// TwinCAT 3 PLC project IntegrationProjects
// Title: IntegrationProjects
// Company: Vortex.Library
// ProjectVersion: 0.6.0.913
// ProgramVersion: 3.1.4023.0
// libraries:
//   Tc2_Standard, * (Beckhoff Automation GmbH)
//   Tc2_System, * (Beckhoff Automation GmbH)
//   Tc3_Module, * (Beckhoff Automation GmbH)
//   TcoCore, 0.6.0.913 (Vortex.Library)
//   TcoData, 0.6.0.913 (Vortex.Library)
//   TcoDrivesBeckhoff, 0.6.0.913 (Vortex.Library)
//   TcoElements, 0.6.0.913 (Vortex.Library)
//   TcoIo, 0.6.0.913 (Vortex.Library)
//   TcoPneumatics, 0.6.0.913 (Vortex.Library)
//   TcoUtilities, 0.6.0.913 (Vortex.Library)
// project tree:
//   / PlcTask.TcTTO
//   POUs/ MAIN.TcPOU, SampleContext.TcPOU
//   POUs/SampleComponent/ SampleComponent.TcPOU, SampleTaskFunctionBuffer.TcDUT, SampleTaskIteration.TcPOU
//   Technology/IO/ EC001.TcDUT, IO.TcGVL
//   Technology/ MAIN_TECHNOLOGY.TcPOU, Technology.TcPOU
//   Technology/ST001/Data/ ST001_ProcessData.TcDUT, ST001_ProcessDataManager.TcPOU
//   Technology/ST001/ ST001.TcPOU, ST001_Components.TcDUT, ST001_ComponentsHandler.TcPOU, ST001_GroundSequence.TcPOU, ST001_AutomatSequence.TcPOU
//   ToLibs/BeckhoffIo/EL1008/ EL1008.TcPOU, EL1008_Data.TcDUT
//   ToLibs/BeckhoffIo/EL2008/ EL2008.TcPOU, EL2008_Data.TcDUT
//   ToLibs/BeckhoffIo/ WcState.TcDUT, InfoData.TcDUT
// real-time tasks:
//   TASK PlcTask: cycle T#10ms, priority 20, ADS port 350
//   TASK PlcTask1: cycle T#10ms, priority 21, ADS port 351
// I/O:
//   DEVICE Device 1 (EtherCAT) (disabled), AmsNetId 172.20.10.104.2.1
//     EC001 (EK1100) [EK1100 EtherCAT Coupler (2A E-Bus)]
//       A1 (EL1008) [EL1008 8Ch. Dig. Input 24V, 3ms]
//       A10 (EL2008) [EL2008 8Ch. Dig. Output 24V, 0.5A]

CONFIGURATION IntegrationProjects
    RESOURCE PLC ON TwinCAT3
        TASK PlcTask(INTERVAL := T#10ms, PRIORITY := 20);
        PROGRAM MAIN WITH PlcTask : MAIN;
        PROGRAM MAIN_TECHNOLOGY WITH PlcTask : MAIN_TECHNOLOGY;
    END_RESOURCE
END_CONFIGURATION

// ---- POUs/SampleComponent/SampleTaskFunctionBuffer.TcDUT
TYPE SampleTaskFunctionBuffer :
    STRUCT
    x : LREAL;
    y : LREAL;
END_STRUCT
END_TYPE

// ---- Technology/IO/EC001.TcDUT
TYPE EC001 :
    STRUCT
    {attribute addProperty Name "A1"}
    A1 : EL1008;
    {attribute addProperty Name "A10"}
    A10 : EL2008;
END_STRUCT
END_TYPE

// ---- Technology/ST001/Data/ST001_ProcessData.TcDUT
TYPE ST001_ProcessData EXTENDS TcoData.TcoEntity :
STRUCT
    PressingTime : TIME;
END_STRUCT
END_TYPE

// ---- Technology/ST001/ST001_Components.TcDUT
TYPE ST001_Components :
    STRUCT
    PartPresent : TcoElements.TcoDi(MAIN_TECHNOLOGY._technology._ST001);
    StartButton : TcoElements.TcoDi(MAIN_TECHNOLOGY._technology._ST001);
    Press : TcoPneumatics.TcoCylinder(MAIN_TECHNOLOGY._technology._ST001);
    Drive : TcoDriveSimple(MAIN_TECHNOLOGY._technology._ST001);
END_STRUCT
END_TYPE

// ---- ToLibs/BeckhoffIo/EL1008/EL1008_Data.TcDUT
TYPE EL1008_Data :
STRUCT
    {attribute addProperty Name "1"}
    _1 AT %I* : BOOL;
    {attribute addProperty Name "2"}
    _2 AT %I* : BOOL;
    {attribute addProperty Name "3"}
    _3 AT %I* : BOOL;
    {attribute addProperty Name "4"}
    _4 AT %I* : BOOL;
    {attribute addProperty Name "5"}
    _5 AT %I* : BOOL;
    {attribute addProperty Name "6"}
    _6 AT %I* : BOOL;
    {attribute addProperty Name "7"}
    _7 AT %I* : BOOL;
    {attribute addProperty Name "7"}
    _8 AT %I* : BOOL;
    WcState : WcState;
    InfoData : InfoData;
END_STRUCT
END_TYPE

// ---- ToLibs/BeckhoffIo/EL2008/EL2008_Data.TcDUT
TYPE EL2008_Data :
STRUCT
    {attribute addProperty Name "1"}
    _1 AT %Q* : BOOL;
    {attribute addProperty Name "2"}
    _2 AT %Q* : BOOL;
    {attribute addProperty Name "3"}
    _3 AT %Q* : BOOL;
    {attribute addProperty Name "4"}
    _4 AT %Q* : BOOL;
    {attribute addProperty Name "5"}
    _5 AT %Q* : BOOL;
    {attribute addProperty Name "6"}
    _6 AT %Q* : BOOL;
    {attribute addProperty Name "7"}
    _7 AT %Q* : BOOL;
    {attribute addProperty Name "8"}
    _8 AT %Q* : BOOL;
    WcState : WcState;
    InfoData : InfoData;
END_STRUCT
END_TYPE

// ---- ToLibs/BeckhoffIo/WcState.TcDUT
TYPE WcState :
STRUCT
    State AT %I* : BOOL;
    InputToggle AT %I* : BOOL;
END_STRUCT
END_TYPE

// ---- ToLibs/BeckhoffIo/InfoData.TcDUT
TYPE InfoData :
STRUCT
    State AT %I* : UINT;
END_STRUCT
END_TYPE

// ---- Technology/IO/IO.TcGVL
{attribute 'qualified_only'}
VAR_GLOBAL
    {attribute addProperty Name "EC001"}
    EC001 : EC001;
END_VAR

// ---- POUs/MAIN.TcPOU
PROGRAM MAIN
VAR
    _sampleContext : SampleContext;
END_VAR

_sampleContext.Run();

END_PROGRAM

// ---- POUs/SampleContext.TcPOU
FUNCTION_BLOCK SampleContext EXTENDS TcoCore.TcoContext
VAR
    _sampleComponent : SampleComponent(THIS^);
END_VAR

(*~
    <docu>
        <summary>
            Main method of the TcoContext. This is the entry point of any control logic that belongs to this context.
            The call of this method is ensured by calling the <c>InstanceName.Run()</c> method, and it must not be called explicitly.
            This method is abstract, and it must be overridden in derived block.
        </summary>
    </docu>
~*)
METHOD PROTECTED Main
_sampleComponent.Service();
_sampleComponent();
END_METHOD

END_FUNCTION_BLOCK

// ---- POUs/SampleComponent/SampleComponent.TcPOU
(*~
    <docu>
        <summary>Sample component for inspiration</summary>
    </docu>
~*)
FUNCTION_BLOCK SampleComponent EXTENDS TcoCore.TcoComponent
VAR
    (*~
        <docu>
            <summary>Counter</summary>
            <remarks>
                > [!IMPORTANT]
                > This member is ignored when rendering.
            </remarks>
        </docu>
    ~*)
    {attribute clr [RenderIgnore()]}
    _counter : INT;
END_VAR
VAR
    (*~
        <docu>
            <summary>Counter</summary>
            <remarks>
                > [!IMPORTANT]
                > This member is readonly.
            </remarks>
        </docu>
    ~*)
    {attribute addProperty Name "Add Result"}
    {attribute clr [ReadOnly()]}
    _addResult : INT;
    {attribute addProperty Name "A"}
    _addNumberOne : INT;
    {attribute addProperty Name "B"}
    _addNumberTwo : INT;
END_VAR
VAR
    _sampleTask : SampleTaskIteration(THIS^);
END_VAR

_addResult := THIS^.AddTwoNumbers(_addNumberOne, _addNumberTwo);
_sampleTask();

(*~
    <docu>
        <summary>Adds two numbers</summary>
        <returns>Sum of two numbers</returns>
    </docu>
~*)
METHOD AddTwoNumbers : INT
VAR_INPUT
    NumberOne : INT;
    NumberTwo : INT;
END_VAR
AddTwoNumbers := NumberOne + NumberTwo;
END_METHOD

{attribute 'TcRpcEnable'}
METHOD INTERNAL AddTwoNumbersTest : INT
VAR_INPUT
    NumberOne : INT;
    NumberTwo : INT;
END_VAR
AddTwoNumbersTest := THIS^.AddTwoNumbers(NumberOne, NumberTwo);
END_METHOD

METHOD FB_init : BOOL
VAR_INPUT
    bInitRetains : BOOL; // if TRUE, the retain variables are initialized (warm start / cold start)
    bInCopyCode : BOOL; // if TRUE, the instance afterwards gets moved into the copy code (online change)
    ParentObject : ITcoObject;
END_VAR
END_METHOD

(*~
    <docu>
        <summary>
            Restores this instance to the Ready state. Can be called explicitly or from within one of the restore mechanisms.
        </summary>
    </docu>
~*)
METHOD Restore : ITcoRestorable
END_METHOD

(*~
    <docu>
        <summary>
            Custom service (manual, maintenance) logic.
            This method must be implemented in derived class.
        </summary>
    </docu>
~*)
METHOD PROTECTED ServiceMode
END_METHOD

METHOD WaitForModulo : BOOL
VAR_INPUT
    Modulo : INT;
END_VAR
_counter := _counter + 1;
WaitForModulo := _counter MOD Modulo = 0;
END_METHOD

{attribute 'TcRpcEnable'}
METHOD INTERNAL WaitForModuloTest : BOOL
VAR_INPUT
    Modulo : INT;
END_VAR
WaitForModuloTest := THIS^.WaitForModulo(Modulo);
END_METHOD

END_FUNCTION_BLOCK

// ---- POUs/SampleComponent/SampleTaskIteration.TcPOU
FUNCTION_BLOCK SampleTaskIteration EXTENDS TcoCore.TcoTask
VAR
    _x : LREAL;
    _y : LREAL;
    _d : LREAL;
    {attribute addProperty Minimum 100}
    {attribute addProperty Maximum 1000}
    _iterations : INT;
    _currentIteration : INT;
END_VAR

IF (Execute()) THEN
    _y := SIN(_x);
    _x := _x + _d;
    _currentIteration := _currentIteration + 1;
    DoneWhen(_currentIteration >= _iterations);
END_IF

METHOD FB_init : BOOL
VAR_INPUT
    bInitRetains : BOOL; // if TRUE, the retain variables are initialized (warm start / cold start)
    bInCopyCode : BOOL; // if TRUE, the instance afterwards gets moved into the copy code (online change)
    ParentObject : ITcoObject;
END_VAR
END_METHOD

(*~
    <docu>
        <summary>
            Restores this instance to the Ready state. Can be called explicitly or from within one of the restore mechanisms.
            <para>
                See also <see cref="PlcDocu.TcoCore.TcoTask.AutoRestorable()"/>
            </para>
        </summary>
    </docu>
~*)
METHOD Restore : ITcoRestorable
SUPER^.Restore();
_x := 0.0;
_y := 0.0;
_currentIteration := 0;
END_METHOD

END_FUNCTION_BLOCK

// ---- Technology/MAIN_TECHNOLOGY.TcPOU
PROGRAM MAIN_TECHNOLOGY
VAR
    _technology : Technology;
END_VAR

_technology.Run();

END_PROGRAM

// ---- Technology/Technology.TcPOU
FUNCTION_BLOCK Technology EXTENDS TcoCore.TcoContext
VAR
    _ST001 : ST001(THIS^);
    _mirrorStartCycle : ULINT;
END_VAR

(*~
    <docu>
        <summary>
            Main method of the TcoContext. This is the entry point of any control logic that belongs to this context.
            The call of this method is ensured by calling the <c>InstanceName.Run()</c> method, and it must not be called explicitly.
            This method is abstract, and it must be overridden in derived block.
        </summary>
    </docu>
~*)
METHOD PROTECTED Main
_ST001();
END_METHOD

END_FUNCTION_BLOCK

// ---- Technology/ST001/ST001.TcPOU
FUNCTION_BLOCK ST001 EXTENDS TcoCore.TcoObject
VAR
    {attribute addProperty Name "<#MANUAL#>"}
    _serviceModeTask : TcoCore.TcoTask(THIS^);
    {attribute addProperty Name "<#GROUND#>"}
    _groundSequenceTask : TcoCore.TcoTask(THIS^);
    {attribute addProperty Name "<#AUTOMAT#>"}
    _automatSequenceTask : TcoCore.TcoTask(THIS^);
    {attribute clr [Container(Layout.Stack)]}
    _components : ST001_ComponentsHandler(THIS^);
    {attribute clr [RenderIgnore()]}
    _mqttMirrorComponents : ST001_ComponentsHandler(THIS^);
    {attribute clr [Container(Layout.Stack)]}
    _groundPositionSequence : ST001_GroundSequence(THIS^, eRestoreMode.None);
    _automatPositionSequence : ST001_AutomatSequence(THIS^, eRestoreMode.None);
    _settings : ST001_ProcessDataManager(THIS^);
    _repository : ST001_ProcessDataManager(THIS^);
END_VAR

_components();
_settings();
_repository();
_groundPositionSequence(inoComponents := _components);
_automatPositionSequence(inoComponents := _components);

IF (_groundSequenceTask.Execute()) THEN
    _serviceModeTask.Abort();
    _groundPositionSequence.Run();
    _groundSequenceTask.DoneWhen(_groundPositionSequence.CurrentStep.ID = _groundPositionSequence.MaxStepID - 1);
END_IF

_automatSequenceTask.Enabled := _groundSequenceTask.Done;

IF (_automatSequenceTask.Execute()) THEN
    _automatPositionSequence.Run();
END_IF

IF (_serviceModeTask.Execute()) THEN
    _automatSequenceTask.Restore();
    _groundSequenceTask.Restore();
    _groundPositionSequence.Restore();
    _components.Service();
END_IF

PROPERTY Repository : REFERENCE TO ST001_ProcessDataManager
GET
Repository REF= _repository;
END_GET
END_PROPERTY

PROPERTY Settings : REFERENCE TO ST001_ProcessDataManager
GET
Settings REF= _settings;
END_GET
END_PROPERTY

END_FUNCTION_BLOCK

// ---- Technology/ST001/ST001_ComponentsHandler.TcPOU
FUNCTION_BLOCK ST001_ComponentsHandler EXTENDS TcoCore.TcoObject
VAR
    ToMirror : STRING;
    {attribute addProperty Name "<#PART PRESENCE SENSOR#>"}
    _partPresent : TcoElements.TcoDi(THIS^);
    {attribute addProperty Name "<#START BUTTON#>"}
    _startButton : TcoElements.TcoDi(THIS^);
    {attribute addProperty Name "<#PRESS PISTON#>"}
    _press : TcoPneumatics.TcoCylinder(THIS^);
    {attribute addProperty Name "<#ALARM OUTPUT#>"}
    _alarmOutput : TcoElements.TcoDo(THIS^);
    {attribute addProperty Name "<#DRIVE#>"}
    _drive : TcoDrivesBeckhoff.TcoDriveSimple(THIS^);
END_VAR

_partPresent(inoSignal := IO.EC001.A1.IO._1);
_startButton(inoSignal := IO.EC001.A1.IO._2);

_press(inoAtHomePos := IO.EC001.A1.IO._3,
    inoAtWorkPos := IO.EC001.A1.IO._4,
    inoToHomePos := IO.EC001.A10.IO._1,
    inoToWorkPos := IO.EC001.A10.IO._2);

PROPERTY PartPresent : REFERENCE TO TcoElements.TcoDi
GET
PartPresent REF= _partPresent;
END_GET
END_PROPERTY

PROPERTY Press : REFERENCE TO TcoPneumatics.TcoCylinder
GET
Press REF= _press;
END_GET
END_PROPERTY

METHOD Service
THIS^._partPresent.Service();
THIS^._startButton.Service();
THIS^._press.Service();
THIS^._alarmOutput.Service();
END_METHOD

END_FUNCTION_BLOCK

// ---- Technology/ST001/ST001_GroundSequence.TcPOU
FUNCTION_BLOCK ST001_GroundSequence EXTENDS TcoCore.TcoSequencer
VAR_IN_OUT
    inoComponents : ST001_ComponentsHandler;
END_VAR

(*~
    <docu>
        <summary>
            Main method of the sequener. Custom code needs to be placed here. The sequencer is executed by call of InstanceName.Run() method.
            This method is abstract, and it must be overridden in derived block.
        </summary>
    </docu>
~*)
METHOD PROTECTED Main : BOOL
IF (NOT __ISVALIDREF(inoComponents)) THEN
    Messenger.Programming('Invalid reference to inoComponents');
    RETURN;
END_IF

IF (Step(inStepID := 100, inEnabled := TRUE, inStepDescription := '<#PRESS IN BASE POSITION#>')) THEN
    //---------------------------------------
    IF (inoComponents.Press.MoveToHome().Done) THEN
        THIS^.CompleteStep();
    END_IF;
    //---------------------------------------
END_IF;

IF (Step(inStepID := 200, inEnabled := TRUE, inStepDescription := '<#CHECK PART REMOVAL FROM THE FIXTURE#>')) THEN
    //---------------------------------------
    IF (inoComponents.PartPresent.IsFalse) THEN
        THIS^.CompleteStep();
    ELSE
        Messenger.Notify('<#Remove part from the fixture please#>');
    END_IF;
    //---------------------------------------
END_IF;

IF (Step(inStepID := MaxStepID - 1, inEnabled := TRUE, inStepDescription := '<#GROUND POSITION COMPLETED#>')) THEN
    //---------------------------------------
    Messenger.Notify('<#Ground position completed; you can start automat sequence.#>');
    //---------------------------------------
END_IF;
END_METHOD

METHOD PROTECTED OnStateChange
VAR_INPUT
    PreviousState : INT;
    NewState : INT;
END_VAR
IF (NOT __ISVALIDREF(inoComponents)) THEN
    RETURN;
END_IF

inoComponents.Press.Restore();
END_METHOD

END_FUNCTION_BLOCK

// ---- Technology/ST001/ST001_AutomatSequence.TcPOU
FUNCTION_BLOCK ST001_AutomatSequence EXTENDS TcoCore.TcoSequencer
VAR_IN_OUT
    inoComponents : ST001_ComponentsHandler;
END_VAR
VAR
    _gTimer_1 : Tc2_Standard.TON;
END_VAR

(*~
    <docu>
        <summary>
            Main method of the sequener. Custom code needs to be placed here. The sequencer is executed by call of InstanceName.Run() method.
            This method is abstract, and it must be overridden in derived block.
        </summary>
    </docu>
~*)
METHOD PROTECTED Main : BOOL
IF (NOT __ISVALIDREF(inoComponents)) THEN
    Messenger.Programming('Invalid reference to inoComponents');
    RETURN;
END_IF

IF (Step(inStepID := 100, inEnabled := TRUE, inStepDescription := '<#LOAD PART INTO FIXTURE#>')) THEN
    //---------------------------------------
    IF (inoComponents.PartPresent.IsTrue) THEN
        THIS^.CompleteStep();
    END_IF;
    //---------------------------------------
END_IF;

IF (Step(inStepID := 200, inEnabled := TRUE, inStepDescription := '<#PRESS START BUTTON TO START OPERATIONS#>')) THEN
    //---------------------------------------
    IF (inoComponents._startButton.IsTrue) THEN
        THIS^.CompleteStep();
    END_IF;
    //---------------------------------------
END_IF;

IF (Step(inStepID := 300, inEnabled := TRUE, inStepDescription := '<#PRESSING#>')) THEN
    //---------------------------------------
    _gTimer_1(IN := inoComponents.Press.MoveToWork().Done, PT := T#500MS);

    IF (_gTimer_1.Q) THEN
        THIS^.CompleteStep();
    END_IF;
    //---------------------------------------
END_IF;

IF (Step(inStepID := 400, inEnabled := TRUE, inStepDescription := '<#MOVING PRESS TO HOME POSITION#>')) THEN
    //---------------------------------------
    IF (inoComponents.Press.MoveToHome().Done) THEN
        THIS^.CompleteStep();
    END_IF;
    //---------------------------------------
END_IF;

IF (Step(inStepID := 500, inEnabled := TRUE, inStepDescription := '<#REMOVE PART FROM THE FIXTURE#>')) THEN
    //---------------------------------------
    IF (inoComponents.PartPresent.IsFalse) THEN
        THIS^.CompleteStep();
    END_IF;
    //---------------------------------------
END_IF;

IF (Step(inStepID := 600, inEnabled := TRUE, inStepDescription := '<#SAVE DATA#>')) THEN
    //---------------------------------------
    IF (THIS^.Station^.Settings.Create(ULINT_TO_STRING(Context.RealTimeClock.TickClock())).Done) THEN
        THIS^.CompleteStep();
    END_IF;
    //---------------------------------------
END_IF;

IF (Step(inStepID := MaxStepID - 1, inEnabled := TRUE, inStepDescription := '<#OPERATIONS COMPLETED#>')) THEN
    //---------------------------------------
    CompleteSequence();
    //---------------------------------------
END_IF;
END_METHOD

METHOD PROTECTED OnStateChange
VAR_INPUT
    PreviousState : INT;
    NewState : INT;
END_VAR
IF (NOT __ISVALIDREF(inoComponents)) THEN
    RETURN;
END_IF

inoComponents.Press.Restore();
_gTimer_1(IN := FALSE);
END_METHOD

PROPERTY Station : POINTER TO ST001
GET
VAR
    refStation : POINTER TO ST001;
END_VAR
IF (__QUERYPOINTER(Parent, refStation)) THEN
    Station := refStation;
END_IF;
END_GET
END_PROPERTY

END_FUNCTION_BLOCK

// ---- Technology/ST001/Data/ST001_ProcessDataManager.TcPOU
FUNCTION_BLOCK ST001_ProcessDataManager EXTENDS TcoData.TcoDataExchange
VAR
    _data : ST001_ProcessData;
END_VAR

SUPER^();

END_FUNCTION_BLOCK

// ---- ToLibs/BeckhoffIo/EL1008/EL1008.TcPOU
FUNCTION_BLOCK EL1008
VAR
    {attribute addProperty Name "CHANNEL_"}
    _io : EL1008_Data;
END_VAR

PROPERTY IO : REFERENCE TO EL1008_Data
GET
IO REF= _io;
END_GET
END_PROPERTY

END_FUNCTION_BLOCK

// ---- ToLibs/BeckhoffIo/EL2008/EL2008.TcPOU
FUNCTION_BLOCK EL2008
VAR
    {attribute addProperty Name "CHANNEL_"}
    _io : EL2008_Data;
END_VAR

PROPERTY IO : REFERENCE TO EL2008_Data
GET
IO REF= _io;
END_GET
END_PROPERTY

END_FUNCTION_BLOCK
